(*******************************************************************************
                          protoc-gen-twincat V0.0.0.0                           
                  https://github.com/TcHaxx/protoc-gen-twincat                  
*******************************************************************************)
{attribute 'no-analysis'}
TYPE ST_RepeatedComplexData :
STRUCT
	complex_data_list : ARRAY[0..4] OF ST_ComplexData;
	complex_data_list_count : UDINT; // Implict generated field for actual number of items in array complex_data_list
END_STRUCT
END_TYPE

(* stored: Version 1.1.0.1
   DUT ST_RepeatedComplexData: Id 8e2308be-f946-405b-a71c-c5ee7b4e65b2 *)
